// TIA Portal V17 export
// export: Created 2025-03-05T08:02:08.5794457Z, ExportSetting WithDefaults, DisplayName Totally Integrated Automation Portal, DisplayVersion V17 Update 8, DisplayName TIA Portal Openness, DisplayVersion V17 Update 8, DisplayName TIA Portal Version Control Interface, DisplayVersion V17, DisplayName SINAMICS Startdrive Advanced, DisplayVersion V17 SP2, DisplayName SINAMICS Startdrive G110M, G120, G120C, G120D, G120P, G115D, DisplayVersion V17 SP2, DisplayName SINAMICS Startdrive G130, G150, S120, S150, SINAMICS MV, S210, DisplayVersion V17 SP2, DisplayName STEP 7 Professional, DisplayVersion V17 Update 8, DisplayName SINUMERIK ONE STEP 7 Toolbox, DisplayVersion V17 Update 12, DisplayName SINUMERIK 840D sl STEP 7 Toolbox, DisplayVersion V17 Update 12, DisplayName STEP 7 Safety, DisplayVersion V17 Update 6, DisplayName WinCC Advanced, DisplayVersion V17 Update 8
TYPE "READ_DATA_MAG"
// stored: IsFailsafeCompliant false
   STRUCT
      FB2_DATA : Struct
         Error : Bool;   // Error
         Done : Bool;   // Done
         Request : Bool;   // Request
         Error_Fault : Bool;   // Error Fault
         Pulse : Bool;   // Pulse
         MAG_POS_IN_NC : Int;   // MAGAZINE POSITION IN NC
         Tool_state : Word;   // Tool state
         TOOL_NUMBER : Int;   // TOOL NUMBER
         MAGAZINE_POSITION : Int;   // MAGAZINE POSITION
      END_STRUCT;
      TOOL_DATA : Struct   // TOOL DATA
         NUM_CUTING_EDGE : Int;   // NUM CUTING EDGE
         QUANTITY_EDGE : Array[1..5] of Real;   // QUANTITY EDGE
         WARNING_EDGE : Array[1..5] of Real;   // WARNING EDGE
         EXPIRED_EDGE : Array[1..5] of Real;   // EXPIRED EDGE
      END_STRUCT;
      PARAM_MAGAZINE : Struct   // PARAM MAGAZINE
         TC_MOP4_QUANTITY_1 : Struct   // TC MOP4 QUANTITY 1
            SYNTAX_ID : Byte := BYTE#16#82;   // SYNTAX ID
            AREA_UNIT : Byte := BYTE#16#81;   // AREA UNIT
            COLUMN : Word := 16#0;   // TOOL NUMBER (HEX) / COLUMN
            LINE : Word := WORD#16#0004;   // $TC_MOP4[TOOL,1] CUTTING REMAINING LIFE COUNTER / LINE
            BLOCKTYPE : Byte := BYTE#16#22;   // BLOCKTYPE
            NUMOFLINE : Byte := BYTE#16#01;   // NUMOFLINE
            DATATYPE : Byte := BYTE#16#0F;   // DATATYPE
            LENGTH : Byte := BYTE#16#08;   // LENGTH
         END_STRUCT;
         TC_MOP4_QUANTITY_2 : Struct   // TC MOP4 QUANTITY 2
            SYNTAX_ID : Byte := BYTE#16#82;   // SYNTAX ID
            AREA_UNIT : Byte := BYTE#16#81;   // AREA UNIT
            COLUMN : Word := 16#0;   // TOOL NUMBER (HEX) / COLUMN
            LINE : Word := WORD#16#000D;   // $TC_MOP4[TOOL,2] CUTTING REMAINING LIFE COUNTER / LINE
            BLOCKTYPE : Byte := BYTE#16#22;   // BLOCKTYPE
            NUMOFLINE : Byte := BYTE#16#01;   // NUMOFLINE
            DATATYPE : Byte := BYTE#16#0F;   // DATATYPE
            LENGTH : Byte := BYTE#16#08;   // LENGTH
         END_STRUCT;
         TC_MOP4_QUANTITY_3 : Struct   // TC MOP4 QUANTITY 3
            SYNTAX_ID : Byte := BYTE#16#82;   // SYNTAX ID
            AREA_UNIT : Byte := BYTE#16#81;   // AREA UNIT
            COLUMN : Word := 16#0;   // TOOL NUMBER (HEX) / COLUMN
            LINE : Word := WORD#16#0016;   // $TC_MOP4[TOOL,3] CUTTING REMAINING LIFE COUNTER / LINE
            BLOCKTYPE : Byte := BYTE#16#22;   // BLOCKTYPE
            NUMOFLINE : Byte := BYTE#16#01;   // NUMOFLINE
            DATATYPE : Byte := BYTE#16#0F;   // DATATYPE
            LENGTH : Byte := BYTE#16#08;   // LENGTH
         END_STRUCT;
         TC_MOP4_QUANTITY_4 : Struct   // TC MOP4 QUANTITY 4
            SYNTAX_ID : Byte := BYTE#16#82;   // SYNTAX ID
            AREA_UNIT : Byte := BYTE#16#81;   // AREA UNIT
            COLUMN : Word := 16#0;   // TOOL NUMBER (HEX) / COLUMN
            LINE : Word := WORD#16#001F;   // $TC_MOP4[TOOL,4] CUTTING REMAINING LIFE COUNTER / LINE
            BLOCKTYPE : Byte := BYTE#16#22;   // BLOCKTYPE
            NUMOFLINE : Byte := BYTE#16#01;   // NUMOFLINE
            DATATYPE : Byte := BYTE#16#0F;   // DATATYPE
            LENGTH : Byte := BYTE#16#08;   // LENGTH
         END_STRUCT;
         TC_MOP4_QUANTITY_5 : Struct   // TC MOP4 QUANTITY 5
            SYNTAX_ID : Byte := BYTE#16#82;   // SYNTAX ID
            AREA_UNIT : Byte := BYTE#16#81;   // AREA UNIT
            COLUMN : Word := 16#0;   // TOOL NUMBER (HEX) / COLUMN
            LINE : Word := WORD#16#0028;   // $TC_MOP4[TOOL,4] CUTTING REMAINING LIFE COUNTER / LINE
            BLOCKTYPE : Byte := BYTE#16#22;   // BLOCKTYPE
            NUMOFLINE : Byte := BYTE#16#01;   // NUMOFLINE
            DATATYPE : Byte := BYTE#16#0F;   // DATATYPE
            LENGTH : Byte := BYTE#16#08;   // LENGTH
         END_STRUCT;
         TC_MOP3_WARNING_1 : Struct   // TC MOP3 WARNING 1
            SYNTAX_ID : Byte := BYTE#16#82;   // SYNTAX ID
            AREA_UNIT : Byte := BYTE#16#81;   // AREA UNIT
            COLUMN : Word := 16#0;   // TOOL NUMBER (HEX) / COLUMN
            LINE : Word := WORD#16#0003;   // $TC_MOP3[TOOL,1] CUTTING PREWARNING LIFE COUNTER / LINE
            BLOCKTYPE : Byte := BYTE#16#22;   // BLOCKTYPE
            NUMOFLINE : Byte := BYTE#16#01;   // NUMOFLINE
            DATATYPE : Byte := BYTE#16#0F;   // DATATYPE
            LENGTH : Byte := BYTE#16#08;   // LENGTH
         END_STRUCT;
         TC_MOP3_WARNING_2 : Struct   // TC MOP3 WARNING 2
            SYNTAX_ID : Byte := BYTE#16#82;   // SYNTAX ID
            AREA_UNIT : Byte := BYTE#16#81;   // AREA UNIT
            COLUMN : Word := 16#0;   // TOOL NUMBER (HEX) / COLUMN
            LINE : Word := WORD#16#000C;   // $TC_MOP3[TOOL,2] CUTTING PREWARNING LIFE COUNTER / LINE
            BLOCKTYPE : Byte := BYTE#16#22;   // BLOCKTYPE
            NUMOFLINE : Byte := BYTE#16#01;   // NUMOFLINE
            DATATYPE : Byte := BYTE#16#0F;   // DATATYPE
            LENGTH : Byte := BYTE#16#08;   // LENGTH
         END_STRUCT;
         TC_MOP3_WARNING_3 : Struct   // TC MOP3 WARNING 3
            SYNTAX_ID : Byte := BYTE#16#82;   // SYNTAX ID
            AREA_UNIT : Byte := BYTE#16#81;   // AREA UNIT
            COLUMN : Word := 16#0;   // TOOL NUMBER (HEX) / COLUMN
            LINE : Word := WORD#16#0015;   // $TC_MOP3[TOOL,3] CUTTING PREWARNING LIFE COUNTER / LINE
            BLOCKTYPE : Byte := BYTE#16#22;   // BLOCKTYPE
            NUMOFLINE : Byte := BYTE#16#01;   // NUMOFLINE
            DATATYPE : Byte := BYTE#16#0F;   // DATATYPE
            LENGTH : Byte := BYTE#16#08;   // LENGTH
         END_STRUCT;
         TC_MOP3_WARNING_4 : Struct   // TC MOP3 WARNING 4
            SYNTAX_ID : Byte := BYTE#16#82;   // SYNTAX ID
            AREA_UNIT : Byte := BYTE#16#81;   // AREA UNIT
            COLUMN : Word := 16#0;   // TOOL NUMBER (HEX) / COLUMN
            LINE : Word := WORD#16#001E;   // $TC_MOP3[TOOL,4] CUTTING PREWARNING LIFE COUNTER / LINE
            BLOCKTYPE : Byte := BYTE#16#22;   // BLOCKTYPE
            NUMOFLINE : Byte := BYTE#16#01;   // NUMOFLINE
            DATATYPE : Byte := BYTE#16#0F;   // DATATYPE
            LENGTH : Byte := BYTE#16#08;   // LENGTH
         END_STRUCT;
         TC_MOP3_WARNING_5 : Struct   // TC MOP3 WARNING 5
            SYNTAX_ID : Byte := BYTE#16#82;   // SYNTAX ID
            AREA_UNIT : Byte := BYTE#16#81;   // AREA UNIT
            COLUMN : Word := 16#0;   // TOOL NUMBER (HEX) / COLUMN
            LINE : Word := WORD#16#0027;   // $TC_MOP3[TOOL,4] CUTTING PREWARNING LIFE COUNTER / LINE
            BLOCKTYPE : Byte := BYTE#16#22;   // BLOCKTYPE
            NUMOFLINE : Byte := BYTE#16#01;   // NUMOFLINE
            DATATYPE : Byte := BYTE#16#0F;   // DATATYPE
            LENGTH : Byte := BYTE#16#08;   // LENGTH
         END_STRUCT;
         TC_MOP13_EXPIRED_1 : Struct   // TC MOP13 EXPIRED 1
            SYNTAX_ID : Byte := BYTE#16#82;   // SYNTAX ID
            AREA_UNIT : Byte := BYTE#16#81;   // AREA UNIT
            COLUMN : Word := 16#0;   // TOOL NUMBER (HEX) / COLUMN
            LINE : Word := WORD#16#0006;   // $TC_MOP13[TOOL,1] CUTTING SET POINT LIFE COUNTER / LINE
            BLOCKTYPE : Byte := BYTE#16#22;   // BLOCKTYPE
            NUMOFLINE : Byte := BYTE#16#01;   // NUMOFLINE
            DATATYPE : Byte := BYTE#16#0F;   // DATATYPE
            LENGTH : Byte := BYTE#16#08;   // LENGTH
         END_STRUCT;
         TC_MOP13_EXPIRED_2 : Struct   // TC MOP13 EXPIRED 2
            SYNTAX_ID : Byte := BYTE#16#82;   // SYNTAX ID
            AREA_UNIT : Byte := BYTE#16#81;   // AREA UNIT
            COLUMN : Word := 16#0;   // TOOL NUMBER (HEX) / COLUMN
            LINE : Word := WORD#16#000F;   // $TC_MOP13[TOOL,2] CUTTING SET POINT LIFE COUNTER / LINE
            BLOCKTYPE : Byte := BYTE#16#22;   // BLOCKTYPE
            NUMOFLINE : Byte := BYTE#16#01;   // NUMOFLINE
            DATATYPE : Byte := BYTE#16#0F;   // DATATYPE
            LENGTH : Byte := BYTE#16#08;   // LENGTH
         END_STRUCT;
         TC_MOP13_EXPIRED_3 : Struct   // TC MOP13 EXPIRED 3
            SYNTAX_ID : Byte := BYTE#16#82;   // SYNTAX ID
            AREA_UNIT : Byte := BYTE#16#81;   // AREA UNIT
            COLUMN : Word := 16#0;   // TOOL NUMBER (HEX) / COLUMN
            LINE : Word := WORD#16#0018;   // $TC_MOP13[TOOL,3] CUTTING SET POINT LIFE COUNTER / LINE
            BLOCKTYPE : Byte := BYTE#16#22;   // BLOCKTYPE
            NUMOFLINE : Byte := BYTE#16#01;   // NUMOFLINE
            DATATYPE : Byte := BYTE#16#0F;   // DATATYPE
            LENGTH : Byte := BYTE#16#08;   // LENGTH
         END_STRUCT;
         TC_MOP13_EXPIRED_4 : Struct   // TC MOP13 EXPIRED 4
            SYNTAX_ID : Byte := BYTE#16#82;   // SYNTAX ID
            AREA_UNIT : Byte := BYTE#16#81;   // AREA UNIT
            COLUMN : Word := 16#0;   // TOOL NUMBER (HEX) / COLUMN
            LINE : Word := WORD#16#0021;   // $TC_MOP13[TOOL,4] CUTTING SET POINT LIFE COUNTER / LINE
            BLOCKTYPE : Byte := BYTE#16#22;   // BLOCKTYPE
            NUMOFLINE : Byte := BYTE#16#01;   // NUMOFLINE
            DATATYPE : Byte := BYTE#16#0F;   // DATATYPE
            LENGTH : Byte := BYTE#16#08;   // LENGTH
         END_STRUCT;
         TC_MOP13_EXPIRED_5 : Struct   // TC MOP13 EXPIRED 5
            SYNTAX_ID : Byte := BYTE#16#82;   // SYNTAX ID
            AREA_UNIT : Byte := BYTE#16#81;   // AREA UNIT
            COLUMN : Word := 16#0;   // TOOL NUMBER (HEX) / COLUMN
            LINE : Word := WORD#16#002A;   // $TC_MOP13[TOOL,4] CUTTING SET POINT LIFE COUNTER / LINE
            BLOCKTYPE : Byte := BYTE#16#22;   // BLOCKTYPE
            NUMOFLINE : Byte := BYTE#16#01;   // NUMOFLINE
            DATATYPE : Byte := BYTE#16#0F;   // DATATYPE
            LENGTH : Byte := BYTE#16#08;   // LENGTH
         END_STRUCT;
      END_STRUCT;
      FB2_VARS : Struct   // FB2 VARS
         TOOL_NUMBER : Struct   // TOOL NUMBER
            error : Bool;   // error
            done : Bool;   // done
            request : Bool;   // request
         END_STRUCT;
         ORIGI_MAGAZINE : Struct   // ORIGI MAGAZINE
            error : Bool;   // error
            done : Bool;   // done
            request : Bool;   // request
         END_STRUCT;
         CUTING_EDGE : Struct   // CUTING EDGE
            error : Bool;   // error
            done : Bool;   // done
            request : Bool;   // request
         END_STRUCT;
         QUANTITY_EDGE : Struct   // QUANTITY EDGE
            error : Bool;   // error
            done : Bool;   // done
            request : Bool;   // request
         END_STRUCT;
         WARNING_EDGE : Struct   // WARNING EDGE
            error : Bool;   // error
            done : Bool;   // done
            request : Bool;   // request
         END_STRUCT;
         EXPIRED_EDGE : Struct   // EXPIRED EDGE
            error : Bool;   // error
            done : Bool;   // done
            request : Bool;   // request
         END_STRUCT;
      END_STRUCT;
      SMNS_PRMTS_MAG : Struct   // SMNS PRMTS MAG
         MAG_DATA_TC_MPP6_PLACE_DATA : Struct   // MAG DATA TC MPP6 PLACE DATA
            SYNTAX_ID : Byte := BYTE#16#82;   // SYNTAX ID
            AREA_UNIT : Byte := BYTE#16#81;   // CHANNEL NUMBER, 81=CH1, 82=CH2 ) / AREA UNIT
            COLUMN : Word := WORD#16#0001;   // MAGAZINE NUMBER / COLUMN
            LINE : Word := 16#0;   // LINE
            BLOCKTYPE : Byte := BYTE#16#28;   // BLOCKTYPE
            NUMOFLINE : Byte := BYTE#16#01;   // NUMOFLINE
            DATATYPE : Byte := BYTE#16#04;   // DATATYPE
            LENGTH : Byte := BYTE#16#02;   // LENGTH
         END_STRUCT;
         MAG_DATA_NUM_CUTTING_EDGES : Struct   // MAG DATA NUM CUTTING EDGES
            SYNTAX_ID : Byte := BYTE#16#82;   // SYNTAX ID
            AREA_UNIT : Byte := BYTE#16#81;   // AREA UNIT
            COLUMN : Word := WORD#16#000E;   // NUM CUTTING EDGES / COLUMN
            LINE : Word := WORD#16#0001;   // LINE
            BLOCKTYPE : Byte := BYTE#16#21;   // BLOCKTYPE
            NUMOFLINE : Byte := BYTE#16#01;   // NUMOFLINE
            DATATYPE : Byte := BYTE#16#04;   // DATATYPE
            LENGTH : Byte := BYTE#16#02;   // LENGTH
         END_STRUCT;
      END_STRUCT;
   END_STRUCT;
   // // TOOL_DATA.QUANTITY_EDGE[1] : QUANTITY EDGE[1]
   // // TOOL_DATA.QUANTITY_EDGE[2] : QUANTITY EDGE[2]
   // // TOOL_DATA.QUANTITY_EDGE[3] : QUANTITY EDGE[3]
   // // TOOL_DATA.QUANTITY_EDGE[4] : QUANTITY EDGE[4]
   // // TOOL_DATA.QUANTITY_EDGE[5] : QUANTITY EDGE[5]
   // // TOOL_DATA.WARNING_EDGE[1] : WARNING EDGE[1]
   // // TOOL_DATA.WARNING_EDGE[2] : WARNING EDGE[2]
   // // TOOL_DATA.WARNING_EDGE[3] : WARNING EDGE[3]
   // // TOOL_DATA.WARNING_EDGE[4] : WARNING EDGE[4]
   // // TOOL_DATA.WARNING_EDGE[5] : WARNING EDGE[5]
   // // TOOL_DATA.EXPIRED_EDGE[1] : EXPIRED EDGE[1]
   // // TOOL_DATA.EXPIRED_EDGE[2] : EXPIRED EDGE[2]
   // // TOOL_DATA.EXPIRED_EDGE[3] : EXPIRED EDGE[3]
   // // TOOL_DATA.EXPIRED_EDGE[4] : EXPIRED EDGE[4]
   // // TOOL_DATA.EXPIRED_EDGE[5] : EXPIRED EDGE[5]
END_TYPE
